FUNCTION_BLOCK LinearMotionLoad (* Model of linear motion with load *)
  (* Standard: 61499-2 *)
  (* Version 1.0, 2011-04-20, Sandeep Patil, The University of Auckland, First build. *)
  (* Compiler header: package fb.rt.pnp; *)
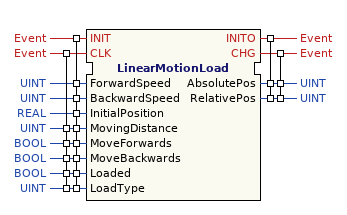
  EVENT_INPUT
    INIT WITH ForwardSpeed, BackwardSpeed, MoveForwards, MoveBackwards, InitialPosition, LoadType, Loaded, MovingDistance; (* Initialization Request *)
    CLK WITH MoveForwards, MoveBackwards, LoadType, Loaded, MovingDistance; (* Clock signal *)
  END_EVENT
  EVENT_OUTPUT
    INITO WITH RelativePos, AbsolutePos; (* Initialization Confirm *)
    CHG WITH RelativePos, AbsolutePos; (* Indicates changes on the data output *)
  END_EVENT
  VAR_INPUT
    ForwardSpeed : UINT; (* Forward speed *)
    BackwardSpeed : UINT; (* Backward speed *)
    InitialPosition : REAL; (* Absolute initial position *)
    MovingDistance : UINT;
    MoveForwards : BOOL; (* Move forwards *)
    MoveBackwards : BOOL; (* Move backwards *)
    Loaded : BOOL;
    LoadType : UINT; (* With different types of load, the actual moving speed varies *)
  END_VAR
  VAR_OUTPUT
    AbsolutePos : UINT;
    RelativePos : UINT; (* Position in percentation *)
  END_VAR
  VAR
    percentagePos : REAL;
  END_VAR
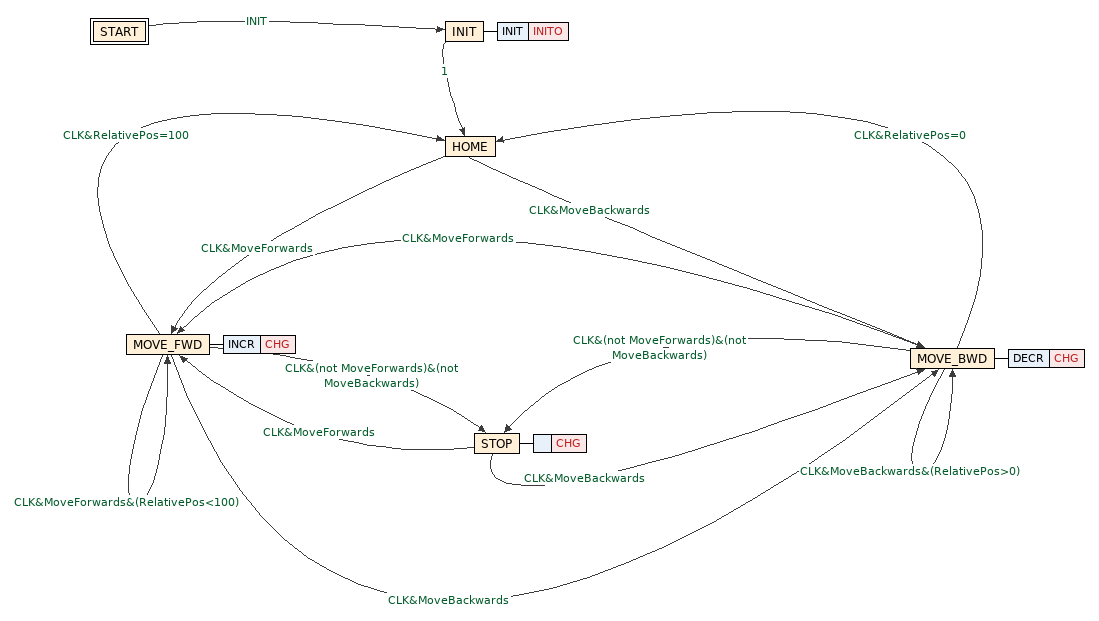
  EC_STATES
    START; (* Initial State *)
    INIT : INIT -> INITO; (* Initialization *)
    MOVE_FWD : INCR -> CHG;
    MOVE_BWD : DECR -> CHG;
    STOP : -> CHG;
    HOME; (* At home position *)
  END_STATES
  EC_TRANSITIONS
    START TO INIT := INIT;
    INIT TO HOME := 1;
    HOME TO MOVE_FWD := CLK&MoveForwards;
    MOVE_FWD TO STOP := CLK&(not MoveForwards)&(not MoveBackwards);
    MOVE_BWD TO STOP := CLK&(not MoveForwards)&(not MoveBackwards);
    STOP TO MOVE_FWD := CLK&MoveForwards;
    STOP TO MOVE_BWD := CLK&MoveBackwards;
    MOVE_BWD TO HOME := CLK&RelativePos=0; (* Back to the home position *)
    MOVE_FWD TO MOVE_BWD := CLK&MoveBackwards;
    MOVE_BWD TO MOVE_FWD := CLK&MoveForwards;
    MOVE_FWD TO MOVE_FWD := CLK&MoveForwards&(RelativePos<100);
    MOVE_BWD TO MOVE_BWD := CLK&MoveBackwards&(RelativePos>0);
    HOME TO MOVE_BWD := CLK&MoveBackwards;
    MOVE_FWD TO HOME := CLK&RelativePos=100;
  END_TRANSITIONS
  ALGORITHM INIT IN Java: (* Initialization algorithm *)
System.out.println("\n  LinearMotion_C.INIT");

float position = (float)InitialPosition.value;

//AbsolutePos.value=(int)Math.ceil(position);
AbsolutePos.value=(int)Math.floor(position);
  END_ALGORITHM
  ALGORITHM INCR IN Java: (* Increment the position *)
// With different types of load, the actual moving speed changes

float position = 0;

// ---------- Check whether the motor is loaded ----------
if(Loaded.value && LoadType.value>0)
{
    position=(float)(AbsolutePos.value+ForwardSpeed.value*(1-LoadType.value/10.0));
    position = (position>MovingDistance.value) ? MovingDistance.value : position;
    percentagePos.value=(int)Math.floor((position/MovingDistance.value)*100);
}
else
{
    position=(float)(AbsolutePos.value+ForwardSpeed.value);
    position = (position>MovingDistance.value) ? MovingDistance.value : position;
    percentagePos.value=(int)Math.floor((position/MovingDistance.value)*100);
}

AbsolutePos.value=(int)Math.floor(position);
RelativePos.value=(int)percentagePos.value;

//System.out.println("PercentagePos = " + RelativePos.value + " " + AbsolutePos.value + " " + position);
  END_ALGORITHM
  ALGORITHM DECR IN Java: (* Decrement the position *)
// ---------- Check whether the motor is loaded ----------

float position = 0;

// ---------- Check whether the motor is loaded ----------
if(Loaded.value && LoadType.value>0)
{
    position=(float)(AbsolutePos.value-BackwardSpeed.value*(1-LoadType.value/10.0));
    position = (position<0) ? 0 : position;
    percentagePos.value=(int)Math.floor((position/MovingDistance.value)*100);
}
else
{
    position=(float)(AbsolutePos.value-BackwardSpeed.value);
    position = (position<0) ? 0 : position;
    percentagePos.value=(int)Math.floor((position/MovingDistance.value)*100);
}

AbsolutePos.value=(int)Math.floor(position);
RelativePos.value=(int)percentagePos.value;
  END_ALGORITHM
END_FUNCTION_BLOCK
